// LS Electric XG5000 project: 동남148
// PLC NewPLC
// module base 0 slot 0: 입출력 모듈:XBC-DN/DP14E (DC 24V 입력 8점, 트랜지스터 출력 6점)

PROGRAM NewProgram (task: 스캔 프로그램)

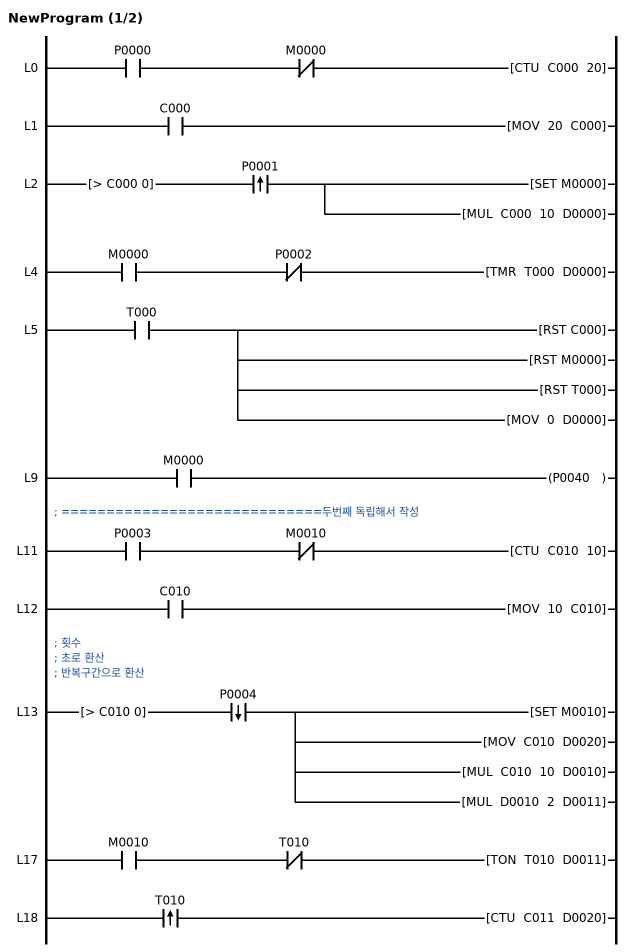
; L0
LOAD      P0000
AND NOT   M0000
CTU       C000 20
; L1
LOAD      C000
MOV       20 C000
; L2
LOAD>     C000 0
ANDP      P0001
SET       M0000
MUL       C000 10 D0000
; L4
LOAD      M0000
AND NOT   P0002
TMR       T000 D0000
; L5
LOAD      T000
RST       C000
RST       M0000
RST       T000
MOV       0 D0000
; L9
LOAD      M0000
OUT       P0040
// =============================두번째 독립해서 작성
; L11
LOAD      P0003
AND NOT   M0010
CTU       C010 10
; L12
LOAD      C010
MOV       10 C010
; L13
LOAD>     C010 0
ANDN      P0004
SET       M0010
MOV       C010 D0020
MUL       C010 10 D0010
MUL       D0010 2 D0011
// output comment: 횟수
// output comment: 초로 환산
// output comment: 반복구간으로 환산
; L17
LOAD      M0010
AND NOT   T010
TON       T010 D0011
; L18
LOADP     T010
CTU       C011 D0020

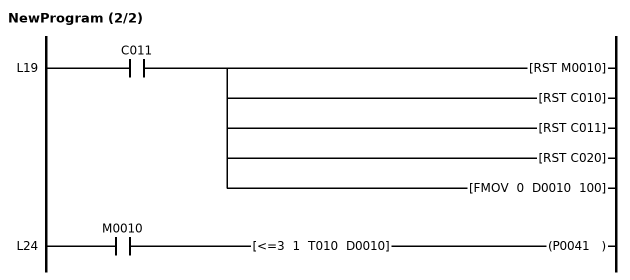
; L19
LOAD      C011
RST       M0010
RST       C010
RST       C011
RST       C020
FMOV      0 D0010 100
; L24
LOAD      M0010
AND<=3    1 T010 D0010
OUT       P0041